(* IEC 61131-3 sources: supports_IUT_Annecy/04_S4/01_POO/01_cours/C02, 2 files *)

(* ---- super_exemple.st ---- *)
FUNCTION_BLOCK FB_1 EXTENDS FB_Base
VAR_OUTPUT
    iBase : INT;
END_VAR

THIS^.METH_DoIt();  //Call of the methods of FB_1
THIS^.METH_DoAlso();

SUPER^.METH_DoIt();   //Call of the methods of FB_Base
SUPER^.METH_DoAlso();
iBase := SUPER^.iCnt;

METHOD METH_DoIt : BOOL
iCnt := 1111;
METH_DoIt := TRUE;

PROGRAM PLC_PRG
VAR
    myBase : FB_Base;
    myFB_1 : FB_1;
    iTHIS : INT;
    iBase : INT;
END_VAR
myBase();
iBase := myBase.iCnt;
myFB_1();
iTHIS := myFB_1.iCnt;

FUNCTION_BLOCK FB_Base
VAR_OUTPUT
    iCnt : INT;
END_VAR

METHOD METH_DoIt : BOOL
iCnt := -1;

METHOD METH_DoAlso : BOOL
METH_DoAlso := TRUE;

FUNCTION_BLOCK FB_1 EXTENDS FB_Base
VAR_OUTPUT
    iBase : INT;
END_VAR

THIS^.METH_DoIt();  //Call of the methods of FB_1
THIS^.METH_DoAlso();

SUPER^.METH_DoIt();   //Call of the methods of FB_Base
SUPER^.METH_DoAlso();
iBase := SUPER^.iCnt;

METHOD METH_DoIt : BOOL
 iCnt := 1111;
 METH_DoIt := TRUE;

PROGRAM PLC_PRG
VAR
 myBase : FB_Base;
 myFB_1 : FB_1;
 iTHIS : INT;
 iBase : INT;
END_VAR

myBase();
iBase := myBase.iCnt;
myFB_1();
iTHIS := myFB_1.iCnt;

(* ---- usercase.st ---- *)
PROGRAM UserCase
VAR
oStep : CStep := (tTaskPeriod := T#10ms);

itfStep : ITF_ObjStep := oStep;
pStep : POINTER TO CStep := ADR(oStep);
xFirstCycleRun : BOOL := TRUE;
END_VAR
IF (xFirstCycleRun) THEN
    ~\dotfill~
    xFirstCycleRun := FALSE;
END_IF
~\dotfill~
~\dotfill~
~\dotfill~
~\dotfill~
